(* Logix 5000 project; controller WWTP_SEC_CLX vendor 1 type 14 code 54 rev 17.2; software revision 17.00; part 2 of 13 *)
(* tags used below, declared in another part *)
   Inp_PVUncertain : BOOL;   // 1=PV Value Not Reliable, 0=OK
   Inp_Sim : BOOL;   // 1=Use simulated PV (Set_SimPV); 0=Use Input (Inp_PV)
   Cfg_NoSubstPV : BOOL;   // 1=Disallow selection of Substitute PV
   Cfg_PCmdClear : BOOL;   // 1=Clear Program Commands on receipt 0=Leave Set
   Cfg_HasHiHiAlm : BOOL;   // 1=High-High Alarm exists and will be checked
   Cfg_HasHiAlm : BOOL;   // 1=High Alarm exists and will be checked
   Cfg_HasLoAlm : BOOL;   // 1=Low Alarm exists and will be checked
   Cfg_HasLoLoAlm : BOOL;   // 1=Low-Low Alarm exists and will be checked
   Cfg_HasFailAlm : BOOL;   // 1=Analog Input Failure Alarm exists and will be checked
   Cfg_FailResetReqd : BOOL;   // 1=Reset required to clear Analog InputFailure Alarm
   Cfg_FailAckReqd : BOOL;   // 1=Acknowledge required for Analog Input Failure Alarm
   Cfg_FailSeverity : SINT;   // Failure Alarm Severity 1=info, 2=warn, 3=excep, 4=fault
   Cfg_HiHiDB : REAL;   // High-High Alarm Deadband (EU)
   Cfg_HiDB : REAL;   // High Alarm Deadband (EU)
   Cfg_LoDB : REAL;   // Low Alarm Deadband (EU)
   Cfg_LoLoDB : REAL;   // Low-Low Alarm Deadband (EU)
   Cfg_FailDB : REAL;   // Out-of-Range (fail) High/Low Deadband (EU)
   Cfg_FailMinDuration : DINT;   // Minimum time Bad or Out of Range to raise Fail Alarm (sec)
   PSet_Owner : DINT;   // Program Owner Request ID (non-zero) or Release (zero)
   PCmd_Acq : BOOL;   // Program Command to Acquire ownership (Oper to Prog)
   PCmd_Rel : BOOL;   // Program Command to Release ownership (Prog to Oper)
   PCmd_Lock : BOOL;   // Program Command to Lock Mode in Prog
   PCmd_Unlock : BOOL;   // Program Command to Unlock Mode
   PCmd_HiHiInhibit : BOOL;   // Program Command to Inhibit High-High Alarm
   PCmd_HiHiUninhibit : BOOL;   // Program Command to UninhibitHigh-High Alarm
   PCmd_HiInhibit : BOOL;   // Program Command to Inhibit High Alarm
   PCmd_HiUninhibit : BOOL;   // Program Command to Uninhibit High Alarm
   PCmd_LoInhibit : BOOL;   // Program Command to Inhibit Low Alarm
   PCmd_LoUninhibit : BOOL;   // Program Command to Uninhibit Low Alarm
   PCmd_LoLoInhibit : BOOL;   // Program Command to Inhibit Low-Low Alarm
   PCmd_LoLoUninhibit : BOOL;   // Program Command to Uninhibit Low-Low Alarm
   PCmd_FailAck : BOOL;   // Program Command to Acknowldege Analog Input Failure Alarm
   PCmd_FailInhibit : BOOL;   // Program Command to Inhibit Analog Input Failure Alarm
   PCmd_FailUninhibit : BOOL;   // Program Command to Uninhibit Analog Input Failure Alarm
   MCmd_SubstPV : BOOL;   // Maintenance Command to use Substitute PV (override input)
   MCmd_InpPV : BOOL;   // Maintenance Command to use Input PV (normal)
   Val_Owner : DINT;   // Current Object Owner ID (0=not owned)
   Sts_SubstPV : BOOL;   // 1=Using Substitute PV (Input being overridden)
   Sts_InpPV : BOOL;   // 1=Using Input PV (normal)
   Sts_PVBad : BOOL;   // 1=PV Bad quality or Out of Range
   Sts_PVUncertain : BOOL;   // 1=PV Value is Uncertain (quality)
   Err_Raw : BOOL;   // 1=Error in Config: Raw Input Scaling Min = Max
   Err_EU : BOOL;   // 1=Error in Config: Scaled EU Min = Max
   Err_Filt : BOOL;   // 1=Error in Config: PV filter params (RateTime, TC)
   Err_DB : BOOL;   // 1=Error in Config: an Alarm Deadband is < 0.0
   Err_Alarm : BOOL;   // 1=Error in Config: Invalid Alarm Min Duration or Severity
   Sts_Maint : BOOL;   // 1=Mode is Maintenance (supersedes Prog, Oper)
   Sts_Prog : BOOL;   // 1=Mode is Program
   Sts_Oper : BOOL;   // 1=Mode is Operator
   Sts_ProgOperLock : BOOL;   // 1=Program or Operator has requested Mode Lock
   Alm_HiHi : BOOL;   // 1=Analog Input is in High-High Alarm
   Ack_HiHi : BOOL;   // 1=High-High Alarm has been acknowledged
   Sts_HiHiDisabled : BOOL;   // 1=High-High Alarm is Disabled (not saved or sent)
   Sts_HiHiInhibited : BOOL;   // 1=High-High Alarm is Inhibited by logic
   Sts_HiHiSuppressed : BOOL;   // 1=High-High Alarm has been suppressed (logged only)
   Alm_Hi : BOOL;   // 1=Analog Input is in High Alarm
   Ack_Hi : BOOL;   // 1=High Alarm has been acknowledged
   Sts_HiDisabled : BOOL;   // 1=High Alarm is Disabled (not saved or sent)
   Sts_HiInhibited : BOOL;   // 1=High Alarm is Inhibited by logic
   Sts_HiSuppressed : BOOL;   // 1=High Alarm has been suppressed (logged only)
   Alm_Lo : BOOL;   // 1=Analog Input is in Low Alarm
   Ack_Lo : BOOL;   // 1=Low Alarm has been acknowledged
   Sts_LoDisabled : BOOL;   // 1=Low Alarm is Disabled (not saved or sent)
   Sts_LoInhibited : BOOL;   // 1=Low Alarm is Inhibited by logic
   Sts_LoSuppressed : BOOL;   // 1=Low Alarm has been suppressed (logged only)
   Alm_LoLo : BOOL;   // 1=Analog Input is in Low-Low Alarm
   Ack_LoLo : BOOL;   // 1=Low-Low Alarm has been acknowledged
   Sts_LoLoDisabled : BOOL;   // 1=Low-Low Alarm is Disabled (not saved or sent)
   Sts_LoLoInhibited : BOOL;   // 1=Low-Low Alarm is Inhibited by logic
   Sts_LoLoSuppressed : BOOL;   // 1=Low-Low Alarm has been suppressed (logged only)
   Sts_Fail : BOOL;   // 1=Analog Input is Out of Range or PV Bad
   Alm_Fail : BOOL;   // 1=Analog Input Failure Alarm (Bad or Out of Range)
   Ack_Fail : BOOL;   // 1=Analog Input Failure Alarm has been acknowledged
   Sts_FailDisabled : BOOL;   // 1=Analog input Failure Alarm is Disabled (not saved or sent)
   Sts_FailInhibited : BOOL;   // 1=Analog Input Failure Alarm is inhibited by logic
   Sts_FailSuppressed : BOOL;   // 1=Analog Input Failure Alarm has been suppressed (logged only)
   Rdy_SubstPV : BOOL;   // 1=Ready for MCmd_SubstPV
   Rdy_InpPV : BOOL;   // 1=Ready for MCmd_InpPV
   LoLo : P_Alarm;   // Low-Low Alarm
   Lo : P_Alarm;   // Low Alarm
   Hi : P_Alarm;   // High Alarm
   HiHi : P_Alarm;   // High-High Alarm
   Mode : P_Mode;   // Analog Input Mode Selection
   Fail : P_Alarm;   // Analog Input Failure Alarm (bad quality or out of range)
   Wrk_Notify : SINT;   // Buffer for building Val_Notify
   Wrk_SubstPV : BOOL;   // Internal flag: Using Substitute PV
   Wrk_ValidONS : BOOL;   // Selected PV goes from Infinite or Not a Number to VALID
   Wrk_SelPVInfNaN : BOOL;   // Selected PV (Input or Substitute) is Infinite or NaN
(* P_AIn, continued *)

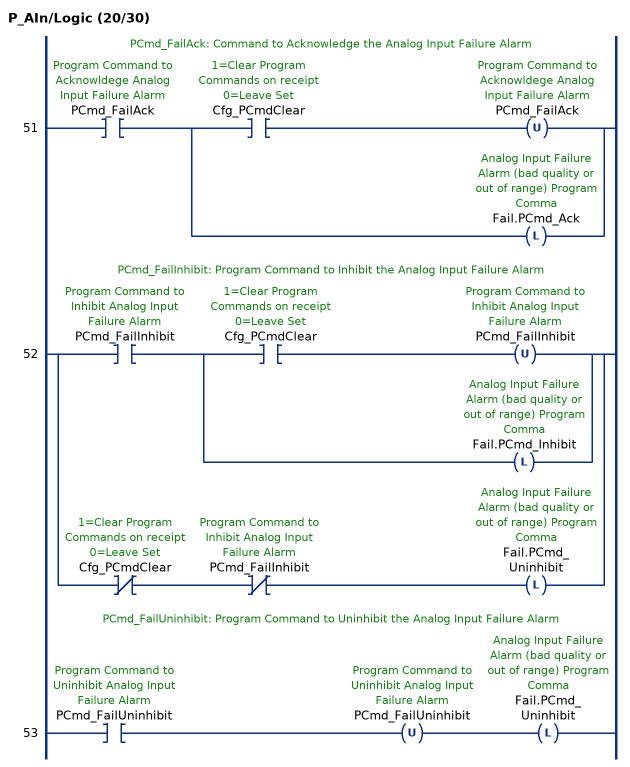
   // PCmd_FailAck: Command to Acknowledge the Analog Input Failure Alarm
   51: XIC(PCmd_FailAck)[XIC(Cfg_PCmdClear) OTU(PCmd_FailAck) ,OTL(Fail.PCmd_Ack) ];
   // PCmd_FailInhibit: Program Command to Inhibit the Analog Input Failure Alarm
   52: [XIC(PCmd_FailInhibit) [XIC(Cfg_PCmdClear) OTU(PCmd_FailInhibit) ,OTL(Fail.PCmd_Inhibit) ] ,XIO(Cfg_PCmdClear) XIO(PCmd_FailInhibit) OTL(Fail.PCmd_Uninhibit) ];
   // PCmd_FailUninhibit: Program Command to Uninhibit the Analog Input Failure Alarm
   53: XIC(PCmd_FailUninhibit)OTU(PCmd_FailUninhibit)OTL(Fail.PCmd_Uninhibit);
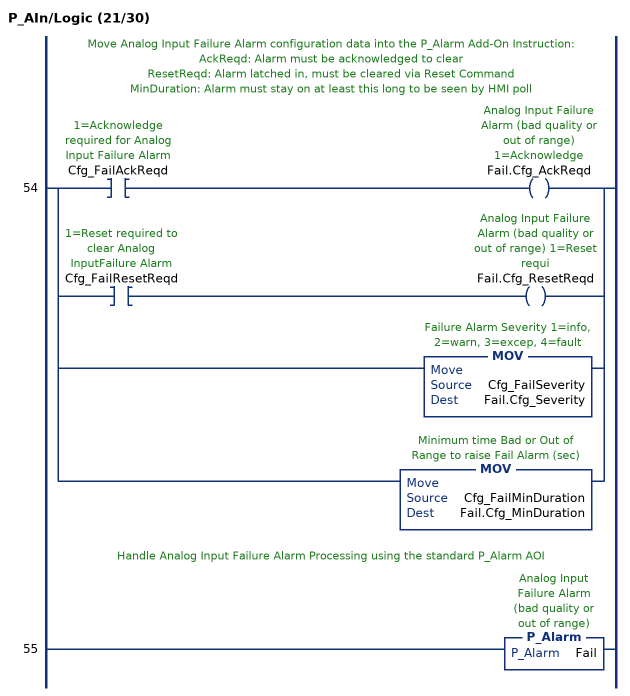
   // Move Analog Input Failure Alarm configuration data into the P_Alarm Add-On Instruction:
   // AckReqd: Alarm must be acknowledged to clear
   // ResetReqd: Alarm latched in, must be cleared via Reset Command
   // MinDuration: Alarm must stay on at least this long to be seen by HMI poll
   54: [XIC(Cfg_FailAckReqd) OTE(Fail.Cfg_AckReqd) ,XIC(Cfg_FailResetReqd) OTE(Fail.Cfg_ResetReqd) ,MOV(Cfg_FailSeverity,Fail.Cfg_Severity) ,MOV(Cfg_FailMinDuration,Fail.Cfg_MinDuration) ];
   // Handle Analog Input Failure Alarm Processing using the standard P_Alarm AOI
   55: P_Alarm(Fail);
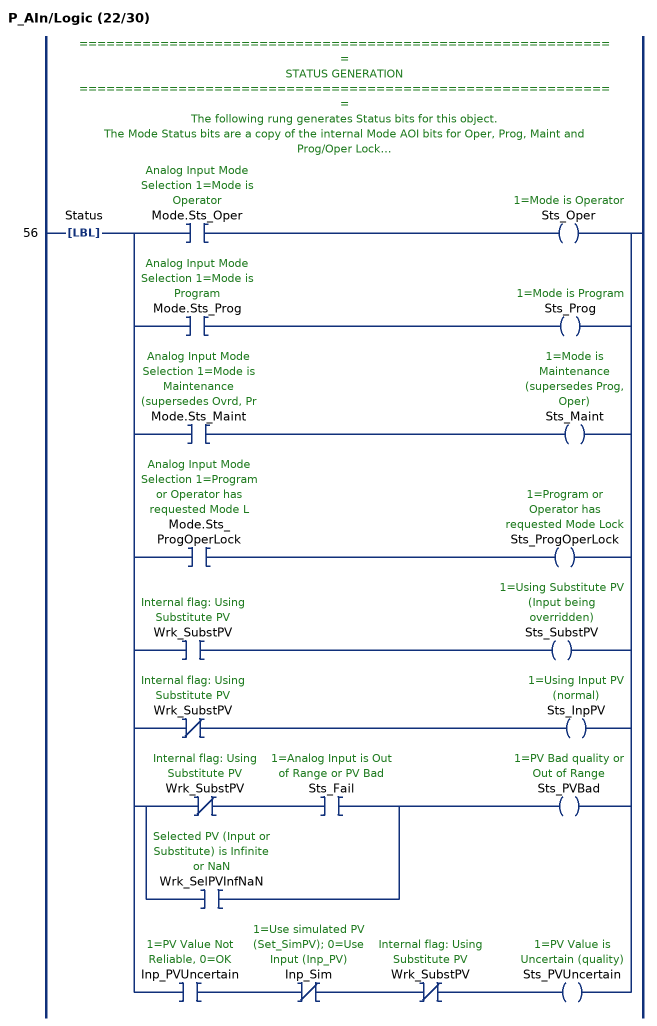
   // ============================================================
   // STATUS GENERATION
   // ============================================================
   // The following rung generates Status bits for this object.
   // The Mode Status bits are a copy of the internal Mode AOI bits for Oper, Prog, Maint and Prog/Oper Lock.
   // Remaining status bits are those not covered in the rungs above.
   56: LBL(Status)[XIC(Mode.Sts_Oper) OTE(Sts_Oper) ,XIC(Mode.Sts_Prog) OTE(Sts_Prog) ,XIC(Mode.Sts_Maint) OTE(Sts_Maint) ,XIC(Mode.Sts_ProgOperLock) OTE(Sts_ProgOperLock) ,XIC(Wrk_SubstPV) OTE(Sts_SubstPV) ,XIO(Wrk_SubstPV) OTE(Sts_InpPV) ,[XIO(Wrk_SubstPV) XIC(Sts_Fail) ,XIC(Wrk_SelPVInfNaN) ] OTE(Sts_PVBad) ,XIC(Inp_PVUncertain) XIO(Inp_Sim) XIO(Wrk_SubstPV) OTE(Sts_PVUncertain) ];
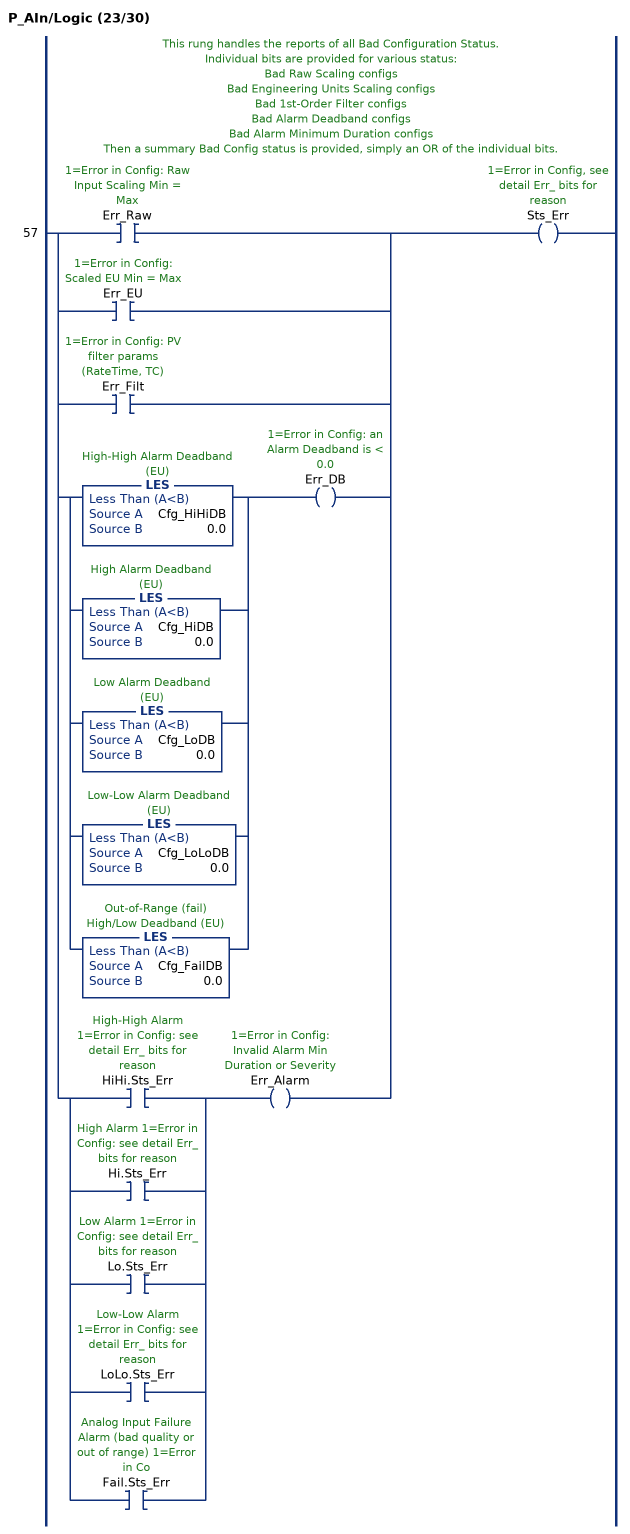
   // This rung handles the reports of all Bad Configuration Status.
   // Individual bits are provided for various status:
   // Bad Raw Scaling configs
   // Bad Engineering Units Scaling configs
   // Bad 1st-Order Filter configs
   // Bad Alarm Deadband configs
   // Bad Alarm Minimum Duration configs
   // Then a summary Bad Config status is provided, simply an OR of the individual bits.
   57: [XIC(Err_Raw) ,XIC(Err_EU) ,XIC(Err_Filt) ,[LES(Cfg_HiHiDB,0.0) ,LES(Cfg_HiDB,0.0) ,LES(Cfg_LoDB,0.0) ,LES(Cfg_LoLoDB,0.0) ,LES(Cfg_FailDB,0.0) ] OTE(Err_DB) ,[XIC(HiHi.Sts_Err) ,XIC(Hi.Sts_Err) ,XIC(Lo.Sts_Err) ,XIC(LoLo.Sts_Err) ,XIC(Fail.Sts_Err) ] OTE(Err_Alarm) ]OTE(Sts_Err);
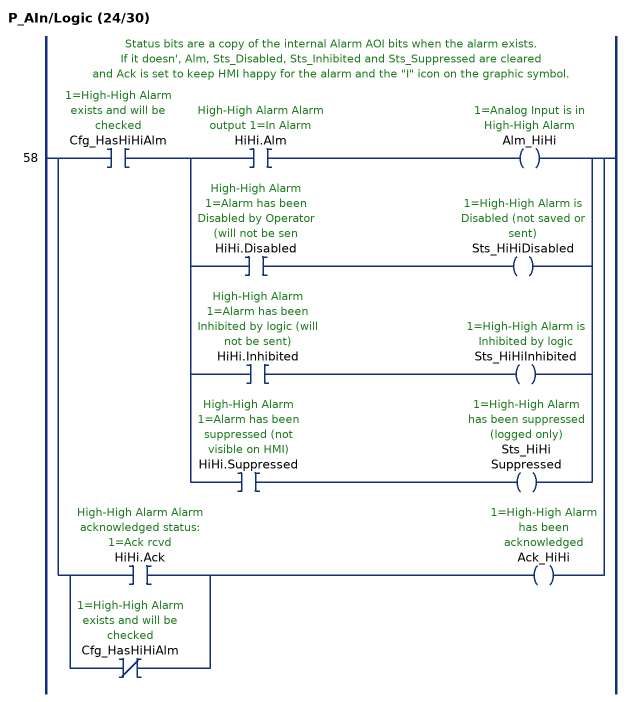
   // Status bits are a copy of the internal Alarm AOI bits when the alarm exists.
   // If it doesn', Alm, Sts_Disabled, Sts_Inhibited and Sts_Suppressed are cleared
   // and Ack is set to keep HMI happy for the alarm and the "I" icon on the graphic symbol.
   58: [XIC(Cfg_HasHiHiAlm) [XIC(HiHi.Alm) OTE(Alm_HiHi) ,XIC(HiHi.Disabled) OTE(Sts_HiHiDisabled) ,XIC(HiHi.Inhibited) OTE(Sts_HiHiInhibited) ,XIC(HiHi.Suppressed) OTE(Sts_HiHiSuppressed) ] ,[XIC(HiHi.Ack) ,XIO(Cfg_HasHiHiAlm) ] OTE(Ack_HiHi) ];
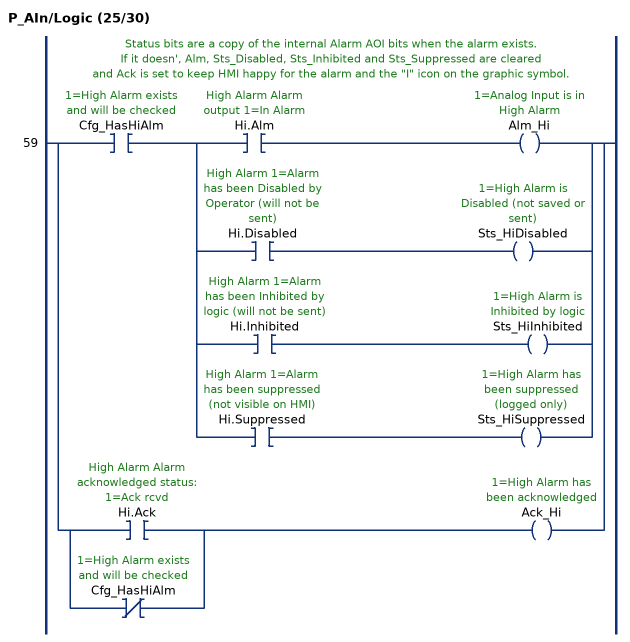
   // Status bits are a copy of the internal Alarm AOI bits when the alarm exists.
   // If it doesn', Alm, Sts_Disabled, Sts_Inhibited and Sts_Suppressed are cleared
   // and Ack is set to keep HMI happy for the alarm and the "I" icon on the graphic symbol.
   59: [XIC(Cfg_HasHiAlm) [XIC(Hi.Alm) OTE(Alm_Hi) ,XIC(Hi.Disabled) OTE(Sts_HiDisabled) ,XIC(Hi.Inhibited) OTE(Sts_HiInhibited) ,XIC(Hi.Suppressed) OTE(Sts_HiSuppressed) ] ,[XIC(Hi.Ack) ,XIO(Cfg_HasHiAlm) ] OTE(Ack_Hi) ];
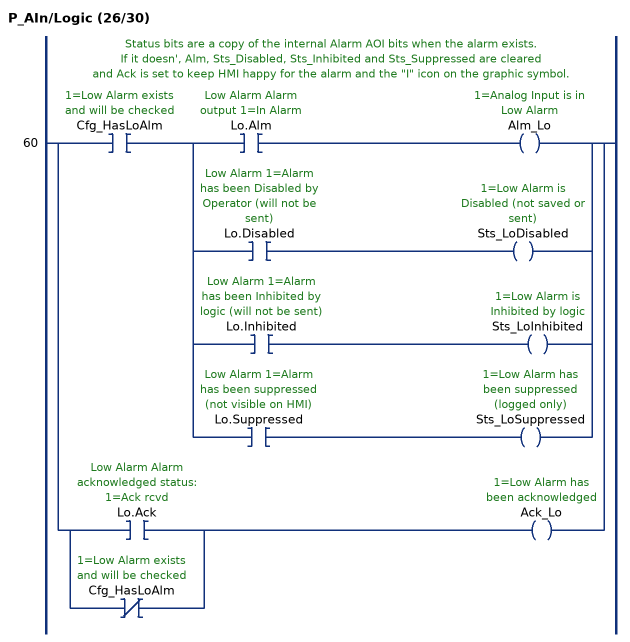
   // Status bits are a copy of the internal Alarm AOI bits when the alarm exists.
   // If it doesn', Alm, Sts_Disabled, Sts_Inhibited and Sts_Suppressed are cleared
   // and Ack is set to keep HMI happy for the alarm and the "I" icon on the graphic symbol.
   60: [XIC(Cfg_HasLoAlm) [XIC(Lo.Alm) OTE(Alm_Lo) ,XIC(Lo.Disabled) OTE(Sts_LoDisabled) ,XIC(Lo.Inhibited) OTE(Sts_LoInhibited) ,XIC(Lo.Suppressed) OTE(Sts_LoSuppressed) ] ,[XIC(Lo.Ack) ,XIO(Cfg_HasLoAlm) ] OTE(Ack_Lo) ];
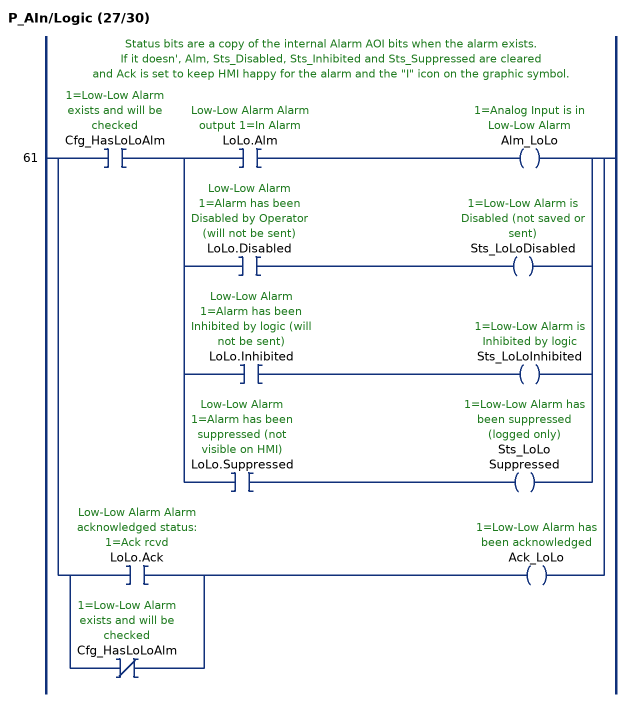
   // Status bits are a copy of the internal Alarm AOI bits when the alarm exists.
   // If it doesn', Alm, Sts_Disabled, Sts_Inhibited and Sts_Suppressed are cleared
   // and Ack is set to keep HMI happy for the alarm and the "I" icon on the graphic symbol.
   61: [XIC(Cfg_HasLoLoAlm) [XIC(LoLo.Alm) OTE(Alm_LoLo) ,XIC(LoLo.Disabled) OTE(Sts_LoLoDisabled) ,XIC(LoLo.Inhibited) OTE(Sts_LoLoInhibited) ,XIC(LoLo.Suppressed) OTE(Sts_LoLoSuppressed) ] ,[XIC(LoLo.Ack) ,XIO(Cfg_HasLoLoAlm) ] OTE(Ack_LoLo) ];
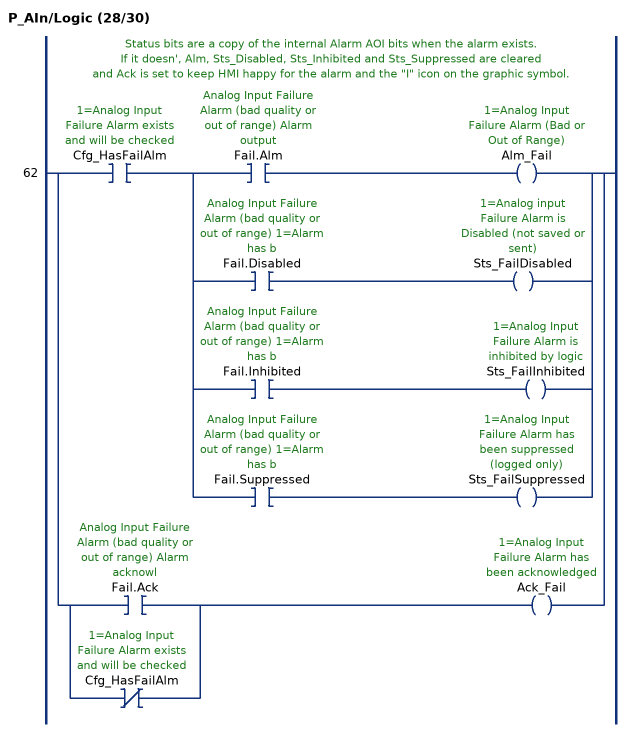
   // Status bits are a copy of the internal Alarm AOI bits when the alarm exists.
   // If it doesn', Alm, Sts_Disabled, Sts_Inhibited and Sts_Suppressed are cleared
   // and Ack is set to keep HMI happy for the alarm and the "I" icon on the graphic symbol.
   62: [XIC(Cfg_HasFailAlm) [XIC(Fail.Alm) OTE(Alm_Fail) ,XIC(Fail.Disabled) OTE(Sts_FailDisabled) ,XIC(Fail.Inhibited) OTE(Sts_FailInhibited) ,XIC(Fail.Suppressed) OTE(Sts_FailSuppressed) ] ,[XIC(Fail.Ack) ,XIO(Cfg_HasFailAlm) ] OTE(Ack_Fail) ];
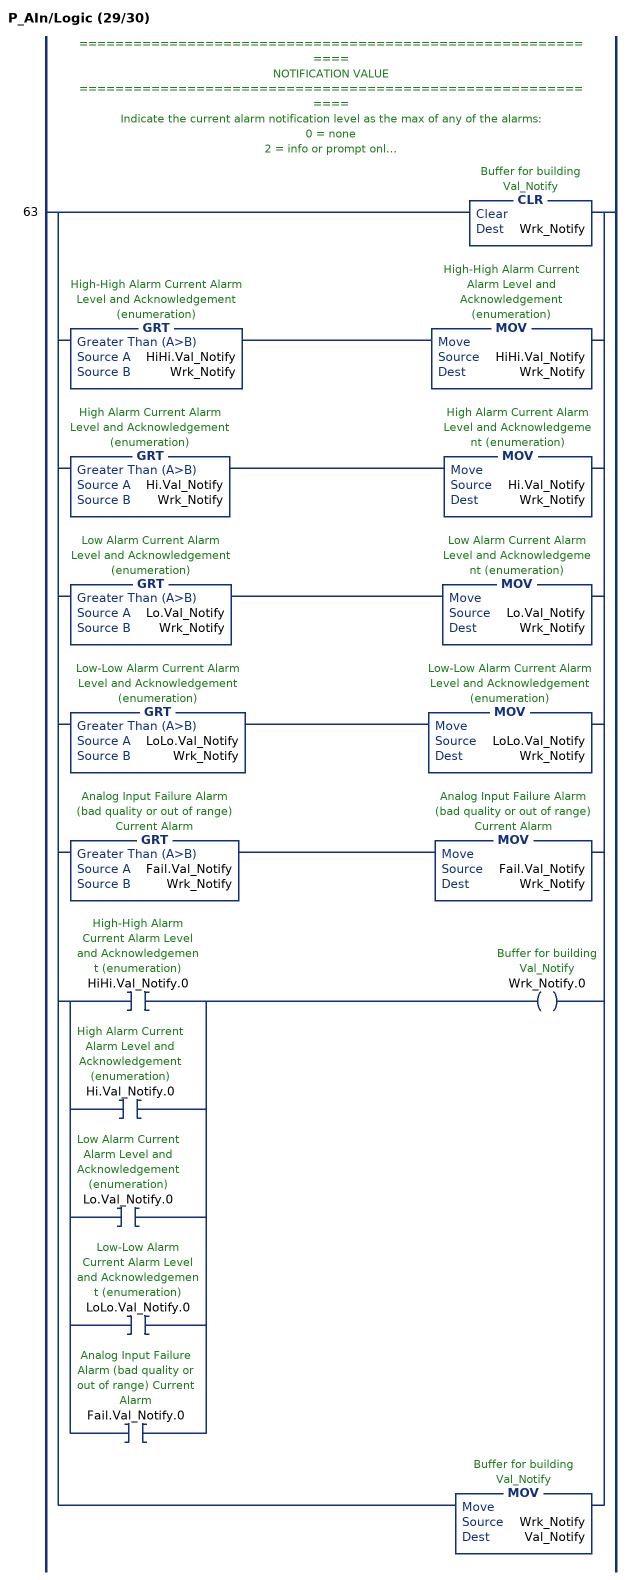
   // ============================================================
   // NOTIFICATION VALUE
   // ============================================================
   // Indicate the current alarm notification level as the max of any of the alarms:
   // 0 = none
   // 2 = info or prompt only
   // 4 = warning
   // 6 = exception (equipment impact)
   // 8 = fault (equipment failure)
   // Add one for any unsuppressed alarm that is not acknowledged (for blink).
   63: [CLR(Wrk_Notify) ,GRT(HiHi.Val_Notify,Wrk_Notify) MOV(HiHi.Val_Notify,Wrk_Notify) ,GRT(Hi.Val_Notify,Wrk_Notify) MOV(Hi.Val_Notify,Wrk_Notify) ,GRT(Lo.Val_Notify,Wrk_Notify) MOV(Lo.Val_Notify,Wrk_Notify) ,GRT(LoLo.Val_Notify,Wrk_Notify) MOV(LoLo.Val_Notify,Wrk_Notify) ,GRT(Fail.Val_Notify,Wrk_Notify) MOV(Fail.Val_Notify,Wrk_Notify) ,[XIC(HiHi.Val_Notify.0) ,XIC(Hi.Val_Notify.0) ,XIC(Lo.Val_Notify.0) ,XIC(LoLo.Val_Notify.0) ,XIC(Fail.Val_Notify.0) ] OTE(Wrk_Notify.0) ,MOV(Wrk_Notify,Val_Notify) ];
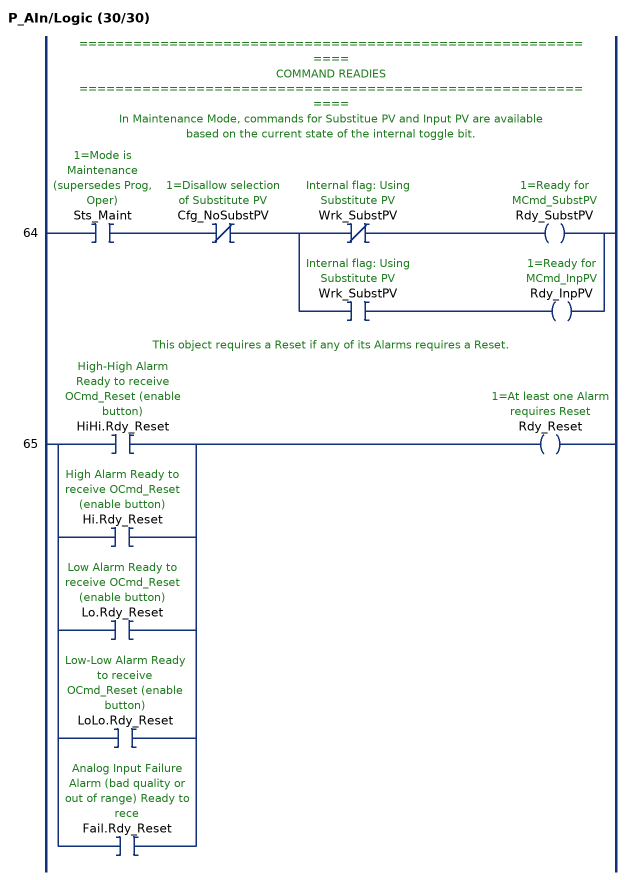
   // ============================================================
   // COMMAND READIES
   // ============================================================
   // In Maintenance Mode, commands for Substitue PV and Input PV are available
   // based on the current state of the internal toggle bit.
   64: XIC(Sts_Maint)XIO(Cfg_NoSubstPV)[XIO(Wrk_SubstPV) OTE(Rdy_SubstPV) ,XIC(Wrk_SubstPV) OTE(Rdy_InpPV) ];
   // This object requires a Reset if any of its Alarms requires a Reset.
   65: [XIC(HiHi.Rdy_Reset) ,XIC(Hi.Rdy_Reset) ,XIC(Lo.Rdy_Reset) ,XIC(LoLo.Rdy_Reset) ,XIC(Fail.Rdy_Reset) ]OTE(Rdy_Reset);
END_ROUTINE

ROUTINE Prescan   (* ladder *)
// Clear Ownership. clear "lurking" Commands
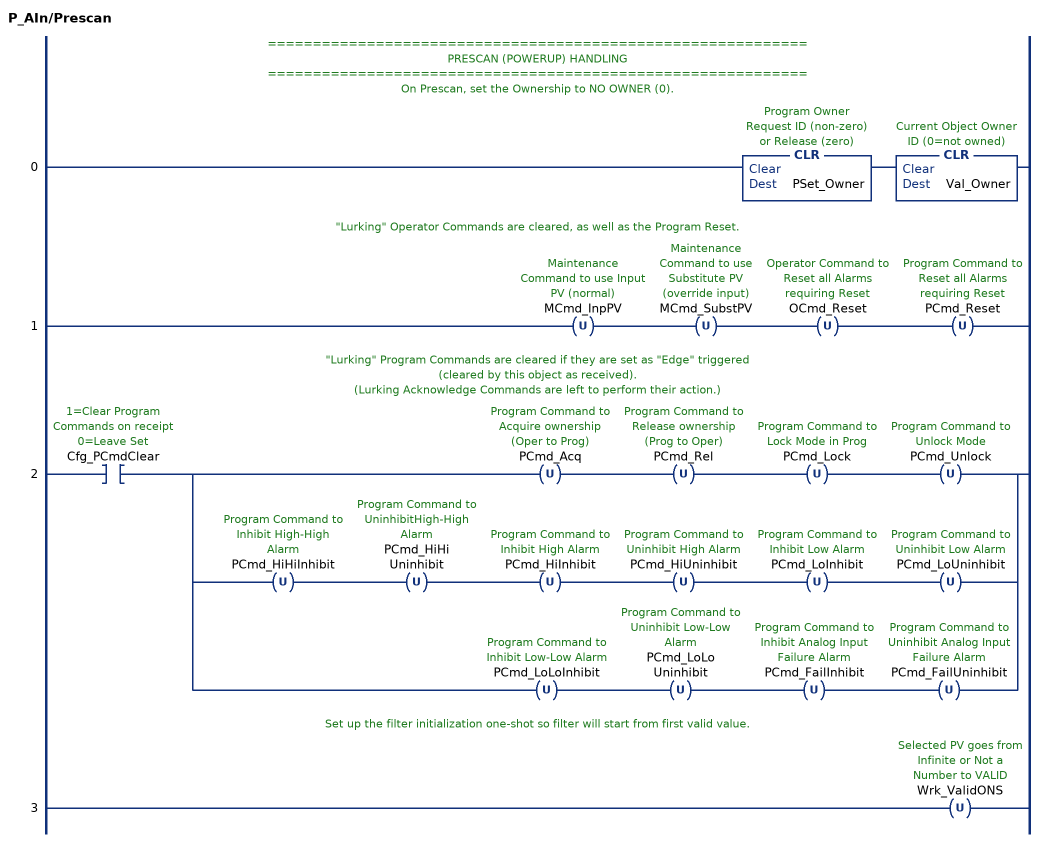
   // ============================================================
   // PRESCAN (POWERUP) HANDLING
   // ============================================================
   // On Prescan, set the Ownership to NO OWNER (0).
   0: CLR(PSet_Owner)CLR(Val_Owner);
   // "Lurking" Operator Commands are cleared, as well as the Program Reset.
   1: OTU(MCmd_InpPV)OTU(MCmd_SubstPV)OTU(OCmd_Reset)OTU(PCmd_Reset);
   // "Lurking" Program Commands are cleared if they are set as "Edge" triggered
   // (cleared by this object as received).
   // (Lurking Acknowledge Commands are left to perform their action.)
   2: XIC(Cfg_PCmdClear)[OTU(PCmd_Acq) OTU(PCmd_Rel) OTU(PCmd_Lock) OTU(PCmd_Unlock) ,OTU(PCmd_HiHiInhibit) OTU(PCmd_HiHiUninhibit) OTU(PCmd_HiInhibit) OTU(PCmd_HiUninhibit) OTU(PCmd_LoInhibit) OTU(PCmd_LoUninhibit) ,OTU(PCmd_LoLoInhibit) OTU(PCmd_LoLoUninhibit) OTU(PCmd_FailInhibit) OTU(PCmd_FailUninhibit) ];
   // Set up the filter initialization one-shot so filter will start from first valid value.
   3: OTU(Wrk_ValidONS);
END_ROUTINE
END_ADD_ON_INSTRUCTION

ADD_ON_INSTRUCTION P_Alarm   (* revision 0.21, ExecutePrescan, ExecuteEnableInFalse *)
// Alarm
// Revision note:
// Fixed differences between Logic and EnableInFalse; fixed scan order dependency.
// Help:
// This instruction monitors one input condition and provides one Alarm with:
//   * configurable Alarm delay, latching, acknowledgement, and severity
//   * commands for enable/disable (oper) and inhibit/uninhibit (prog)
//   * FTA&E suppress/unsuppress support
// This instruction is usually nested within other instructions, with one instance used for each Alarm generated by the containing instruction.  It may also be used as a standalone instruction for Alarm conditions generated by custom logic.
VAR_INPUT
   Inp : BOOL := 1; {visible}   // Alarm Condition Input 1=Alarm
   Inp_Reset : BOOL; {visible}   // 1=Reset Alarm requiring reset
   Cfg_ResetReqd : BOOL;   // 1=Reset required to clear Alarm
   Cfg_AckReqd : BOOL := 1;   // 1=Acknowledge required for Alarm
   Cfg_Severity : SINT := 3;   // 1=Info Only; 2=Warning; 3=Process Exception; 4=Fault
   Cfg_MinDuration : DINT;   // Minimum time (sec) Input must stay on to generate Alarm
   PCmd_Reset : BOOL;   // Program Command to Reset latched alarm
   PCmd_Ack : BOOL;   // Program Command to Acknowledge alarm
   PCmd_Inhibit : BOOL;   // Program Command to Inhibit alarm (force Alm to 0)
   PCmd_Uninhibit : BOOL;   // Program Command to Uninhibit alarm
   OCmd_Reset : BOOL;   // Operator Command to Reset latched alarm
   OCmd_Ack : BOOL;   // Operator Command to Acknowledge alarm
   OCmd_Disable : BOOL;   // Operator Command to Disable alarm (force Alm to 0)
   OCmd_Enable : BOOL;   // Operator Command to Enable alarm
END_VAR
VAR_OUTPUT
   Val_Notify : SINT;   // Current Alarm Level and Acknowledgement (enumeration)
   Alm : BOOL; {visible}   // Alarm output 1=In Alarm
   Ack : BOOL := 1; {visible}   // Alarm acknowledged status: 1=Ack rcvd
   Disabled : BOOL; {visible}   // 1=Alarm has been Disabled by Operator (will not be sent)
   Inhibited : BOOL; {visible}   // 1=Alarm has been Inhibited by logic (will not be sent)
   Suppressed : BOOL; {visible}   // 1=Alarm has been suppressed (not visible on HMI)
   Sts_Err : BOOL;   // 1=Error in Config: see detail Err_ bits for reason
   Err_MinDuration : BOOL;   // 1=Error in Config: Invalid Min Duration (use 0 to 2147483)
   Err_Severity : BOOL;   // 1=Error in Config: Invalid Severity (use 1 to 4)
   Rdy_Reset : BOOL;   // Ready to receive OCmd_Reset (enable button)
   Rdy_Ack : BOOL;   // Ready to receive OCmd_Ack (enable button)
   Rdy_Disable : BOOL := 1;   // Ready to receive OCmd_Disable (enable button)
   Rdy_Enable : BOOL;   // Ready to receive OCmd_Enable (enable button)
END_VAR
VAR
   Wrk_MinDurationT : TIMER;   // Alarm Condition Minimum Duration Timer
   Wrk_Alm : BOOL;   // Internal Alarm Status
   Wrk_Inhibited : BOOL;   // Internal Alarm Inhibit Status
   Wrk_AlmMinOnT : TIMER := (PRE := 5000);   // Alarm output minimum ON time to be seen by alarm server
END_VAR

ROUTINE EnableInFalse   (* ladder *)
// Perform Alarm processing, but Invert Alarm Input ("Inp") for use on LD rung (EnableIn False)
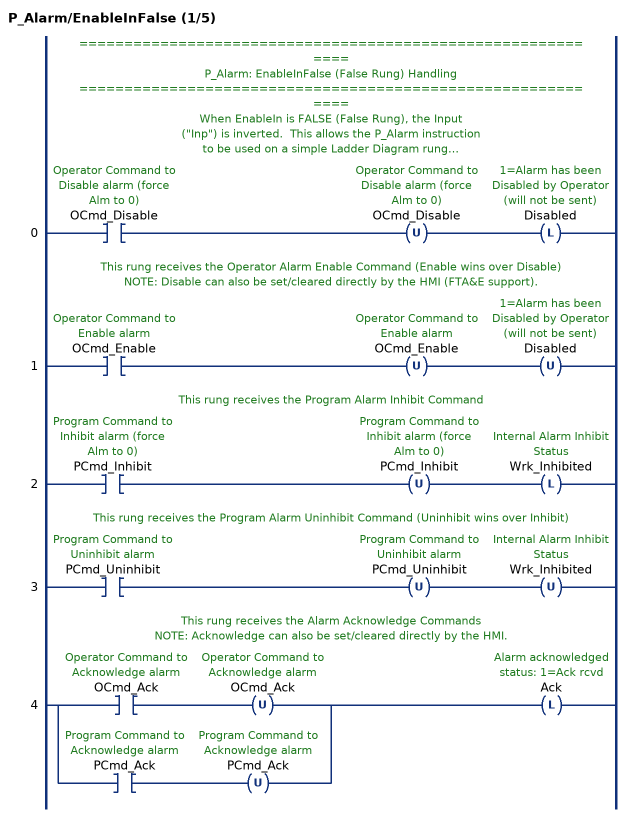
   // ============================================================
   // P_Alarm: EnableInFalse (False Rung) Handling
   // ============================================================
   // When EnableIn is FALSE (False Rung), the Input
   // ("Inp") is inverted.  This allows the P_Alarm instruction
   // to be used on a simple Ladder Diagram rung:
   // XIC  (condition)   P_Alarm (Alarm)
   // All processing is identical to the normal Logic
   // routine, except references to Inp are inverted!
   // ============================================================
   // COMMAND PROCESSING
   // ============================================================
   // These rungs handle received Commands:
   // Operator Commands (OCmd_xx) from the HMI and
   // Program Command (PCmd_xx) from other objects.
   // NOTE:  ALARM COMMANDS ARE ACCEPTED REGARDLESS OF MODE.
   // This rung receives the Operator Alarm Disable Command
   0: XIC(OCmd_Disable)OTU(OCmd_Disable)OTL(Disabled);
   // This rung receives the Operator Alarm Enable Command (Enable wins over Disable)
   // NOTE: Disable can also be set/cleared directly by the HMI (FTA&E support).
   1: XIC(OCmd_Enable)OTU(OCmd_Enable)OTU(Disabled);
   // This rung receives the Program Alarm Inhibit Command
   2: XIC(PCmd_Inhibit)OTU(PCmd_Inhibit)OTL(Wrk_Inhibited);
   // This rung receives the Program Alarm Uninhibit Command (Uninhibit wins over Inhibit)
   3: XIC(PCmd_Uninhibit)OTU(PCmd_Uninhibit)OTU(Wrk_Inhibited);
   // This rung receives the Alarm Acknowledge Commands
   // NOTE: Acknowledge can also be set/cleared directly by the HMI.
   4: [XIC(OCmd_Ack) OTU(OCmd_Ack) ,XIC(PCmd_Ack) OTU(PCmd_Ack) ]OTL(Ack);
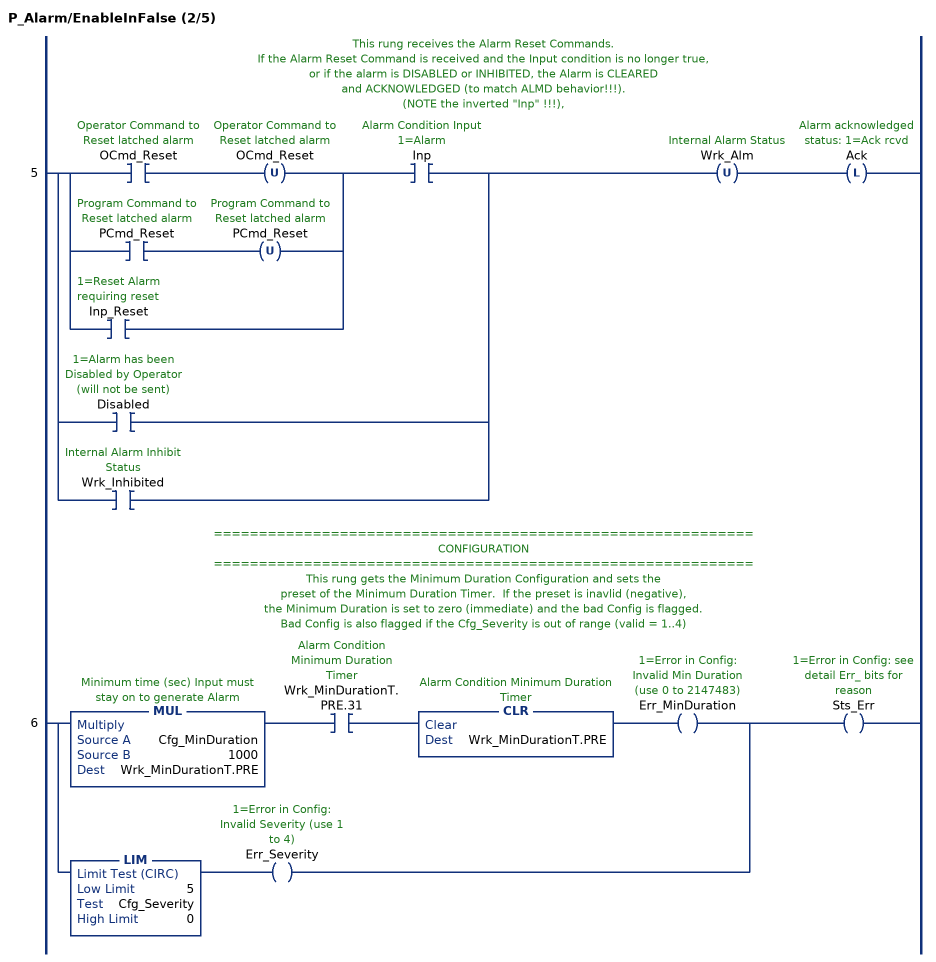
   // This rung receives the Alarm Reset Commands.
   // If the Alarm Reset Command is received and the Input condition is no longer true,
   // or if the alarm is DISABLED or INHIBITED, the Alarm is CLEARED
   // and ACKNOWLEDGED (to match ALMD behavior!!!).
   // (NOTE the inverted "Inp" !!!),
   5: [[XIC(OCmd_Reset) OTU(OCmd_Reset) ,XIC(PCmd_Reset) OTU(PCmd_Reset) ,XIC(Inp_Reset) ] XIC(Inp) ,XIC(Disabled) ,XIC(Wrk_Inhibited) ]OTU(Wrk_Alm)OTL(Ack);
   // ============================================================
   // CONFIGURATION
   // ============================================================
   // This rung gets the Minimum Duration Configuration and sets the
   // preset of the Minimum Duration Timer.  If the preset is inavlid (negative),
   // the Minimum Duration is set to zero (immediate) and the bad Config is flagged.
   // Bad Config is also flagged if the Cfg_Severity is out of range (valid = 1..4)
   6: [MUL(Cfg_MinDuration,1000,Wrk_MinDurationT.PRE) XIC(Wrk_MinDurationT.PRE.31) CLR(Wrk_MinDurationT.PRE) OTE(Err_MinDuration) ,LIM(5,Cfg_Severity,0) OTE(Err_Severity) ]OTE(Sts_Err);
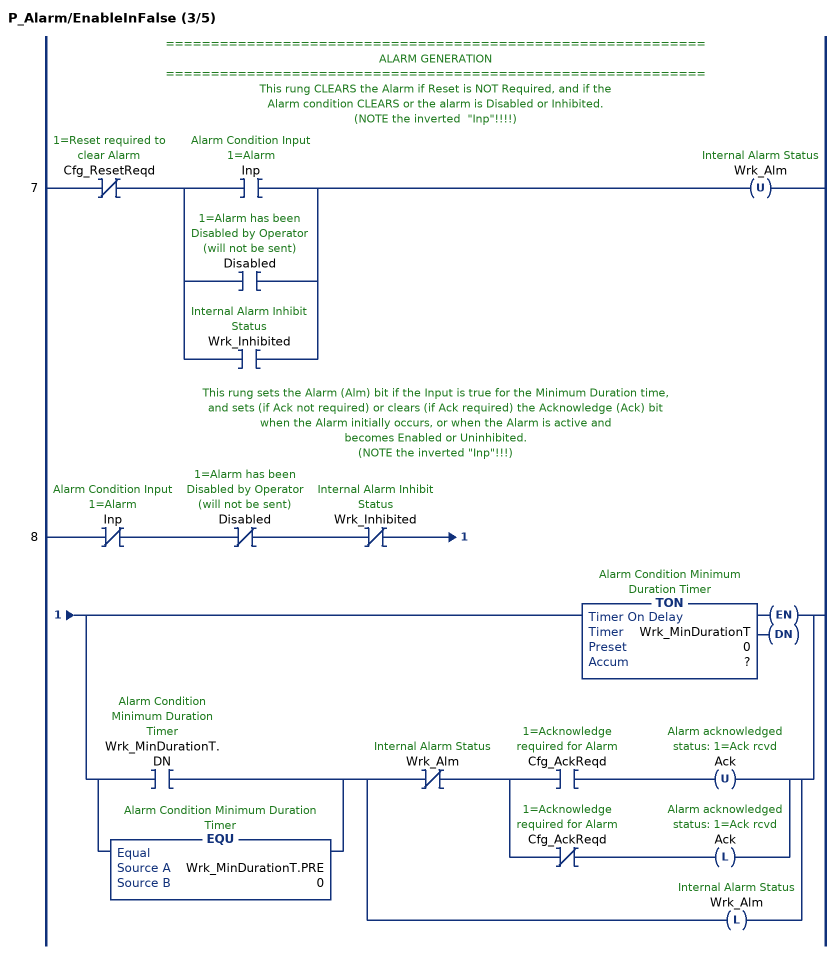
   // ============================================================
   // ALARM GENERATION
   // ============================================================
   // This rung CLEARS the Alarm if Reset is NOT Required, and if the
   // Alarm condition CLEARS or the alarm is Disabled or Inhibited.
   // (NOTE the inverted  "Inp"!!!!)
   7: XIO(Cfg_ResetReqd)[XIC(Inp) ,XIC(Disabled) ,XIC(Wrk_Inhibited) ]OTU(Wrk_Alm);
   // This rung sets the Alarm (Alm) bit if the Input is true for the Minimum Duration time,
   // and sets (if Ack not required) or clears (if Ack required) the Acknowledge (Ack) bit
   // when the Alarm initially occurs, or when the Alarm is active and
   // becomes Enabled or Uninhibited.
   // (NOTE the inverted "Inp"!!!)
   8: XIO(Inp)XIO(Disabled)XIO(Wrk_Inhibited)[TON(Wrk_MinDurationT,?,?) ,[XIC(Wrk_MinDurationT.DN) ,EQU(Wrk_MinDurationT.PRE,0) ] [XIO(Wrk_Alm) [XIC(Cfg_AckReqd) OTU(Ack) ,XIO(Cfg_AckReqd) OTL(Ack) ] ,OTL(Wrk_Alm) ] ];
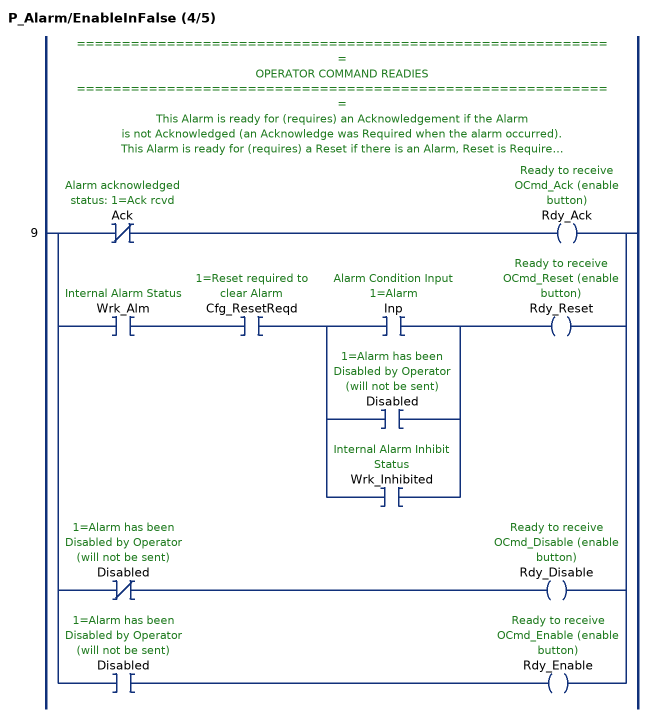
   // ============================================================
   // OPERATOR COMMAND READIES
   // ============================================================
   // This Alarm is ready for (requires) an Acknowledgement if the Alarm
   // is not Acknowledged (an Acknowledge was Required when the alarm occurred).
   // This Alarm is ready for (requires) a Reset if there is an Alarm, Reset is Required
   // and the Alarm Condition is CLEARED
   // (NOTE the inverted "Inp"!!!)
   // If the Alarm is NOT Disabled, it is ready for Disable.
   // If the Alarm IS Disabled, it is ready for Enable.
   9: [XIO(Ack) OTE(Rdy_Ack) ,XIC(Wrk_Alm) XIC(Cfg_ResetReqd) [XIC(Inp) ,XIC(Disabled) ,XIC(Wrk_Inhibited) ] OTE(Rdy_Reset) ,XIO(Disabled) OTE(Rdy_Disable) ,XIC(Disabled) OTE(Rdy_Enable) ];
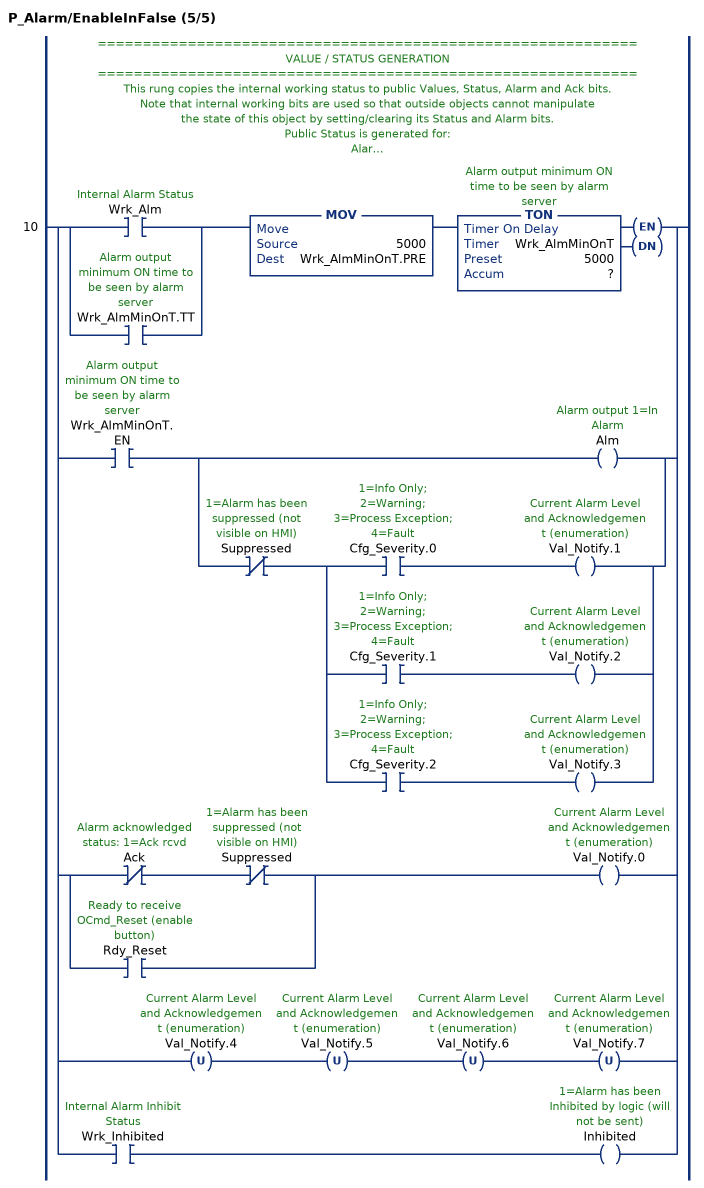
   // ============================================================
   // VALUE / STATUS GENERATION
   // ============================================================
   // This rung copies the internal working status to public Values, Status, Alarm and Ack bits.
   // Note that internal working bits are used so that outside objects cannot manipulate
   // the state of this object by setting/clearing its Status and Alarm bits.
   // Public Status is generated for:
   // Alarm
   // Notify Level (color, blink)
   // Alarm Inhibited
   // (Ack, Suppressed and Disabled can be set/cleared by the HMI directly.)
   10: [[XIC(Wrk_Alm) ,XIC(Wrk_AlmMinOnT.TT) ] MOV(5000,Wrk_AlmMinOnT.PRE) TON(Wrk_AlmMinOnT,?,?) ,XIC(Wrk_AlmMinOnT.EN) [OTE(Alm) ,XIO(Suppressed) [XIC(Cfg_Severity.0) OTE(Val_Notify.1) ,XIC(Cfg_Severity.1) OTE(Val_Notify.2) ,XIC(Cfg_Severity.2) OTE(Val_Notify.3) ] ] ,[XIO(Ack) XIO(Suppressed) ,XIC(Rdy_Reset) ] OTE(Val_Notify.0) ,OTU(Val_Notify.4) OTU(Val_Notify.5) OTU(Val_Notify.6) OTU(Val_Notify.7) ,XIC(Wrk_Inhibited) OTE(Inhibited) ];
END_ROUTINE

ROUTINE Logic   (* ladder *)
// Perform Alarm processing: delay, latch/reset, acknowledge, enable/disable, inhibit/uninhibit, suppress/unsuppress
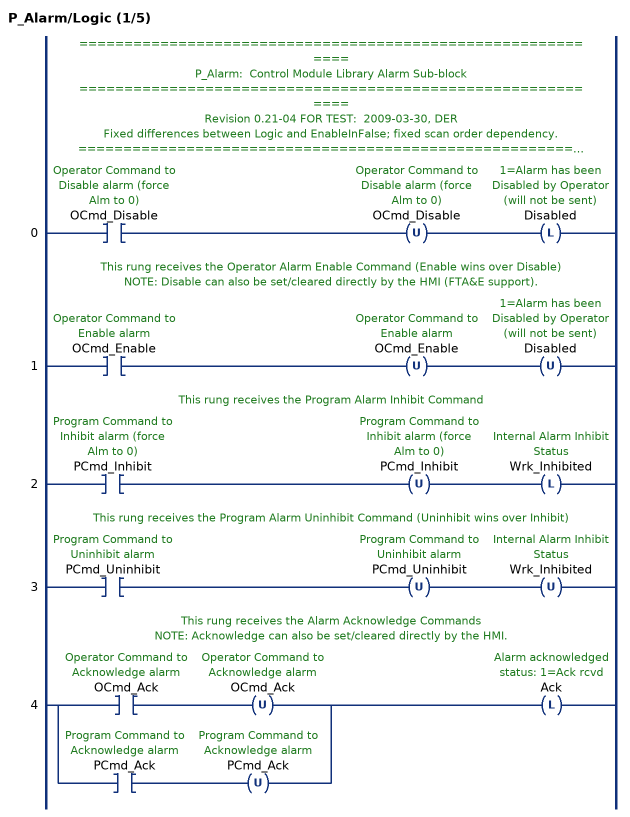
   // ============================================================
   // P_Alarm:  Control Module Library Alarm Sub-block
   // ============================================================
   // Revision 0.21-04 FOR TEST:  2009-03-30, DER
   // Fixed differences between Logic and EnableInFalse; fixed scan order dependency.
   // ============================================================
   // This instruction provides standard Alarm handling for a given input Alarm condition.
   // This instruction should be imbedded in any instruction that generates alarms,
   // one instance per alarm generated.
   // ============================================================
   // POWERUP / INVALID STATE HANDLING
   // ============================================================
   // All internal Work (state) bits maintain states through a power cycle and are
   // independent.  No first-scan logic is required.  See the Prescan routine for
   // powerup / prescan code.
   // ============================================================
   // COMMAND PROCESSING
   // ============================================================
   // These rungs handle received Commands:
   // Operator Commands (OCmd_xx) from the HMI and
   // Program Command (PCmd_xx) from other objects.
   // NOTE:  ALARM COMMANDS ARE ACCEPTED REGARDLESS OF MODE.
   // This rung receives the Operator Alarm Disable Command
   0: XIC(OCmd_Disable)OTU(OCmd_Disable)OTL(Disabled);
   // This rung receives the Operator Alarm Enable Command (Enable wins over Disable)
   // NOTE: Disable can also be set/cleared directly by the HMI (FTA&E support).
   1: XIC(OCmd_Enable)OTU(OCmd_Enable)OTU(Disabled);
   // This rung receives the Program Alarm Inhibit Command
   2: XIC(PCmd_Inhibit)OTU(PCmd_Inhibit)OTL(Wrk_Inhibited);
   // This rung receives the Program Alarm Uninhibit Command (Uninhibit wins over Inhibit)
   3: XIC(PCmd_Uninhibit)OTU(PCmd_Uninhibit)OTU(Wrk_Inhibited);
   // This rung receives the Alarm Acknowledge Commands
   // NOTE: Acknowledge can also be set/cleared directly by the HMI.
   4: [XIC(OCmd_Ack) OTU(OCmd_Ack) ,XIC(PCmd_Ack) OTU(PCmd_Ack) ]OTL(Ack);
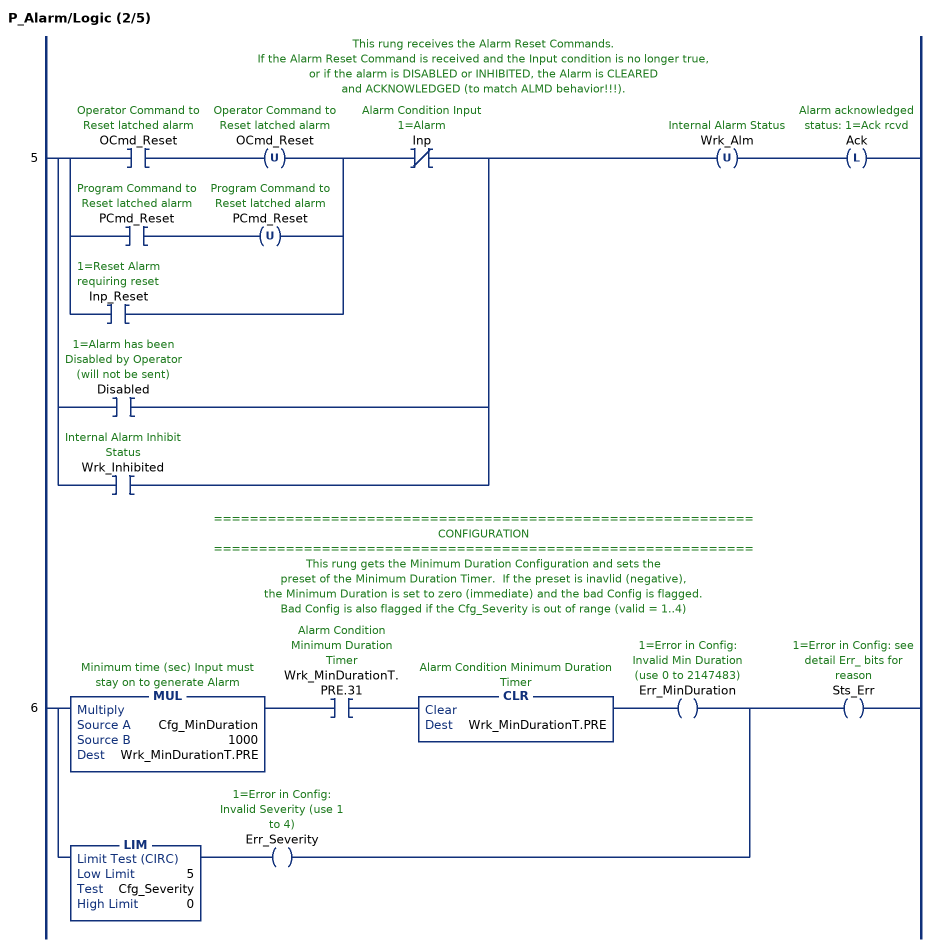
   // This rung receives the Alarm Reset Commands.
   // If the Alarm Reset Command is received and the Input condition is no longer true,
   // or if the alarm is DISABLED or INHIBITED, the Alarm is CLEARED
   // and ACKNOWLEDGED (to match ALMD behavior!!!).
   5: [[XIC(OCmd_Reset) OTU(OCmd_Reset) ,XIC(PCmd_Reset) OTU(PCmd_Reset) ,XIC(Inp_Reset) ] XIO(Inp) ,XIC(Disabled) ,XIC(Wrk_Inhibited) ]OTU(Wrk_Alm)OTL(Ack);
   // ============================================================
   // CONFIGURATION
   // ============================================================
   // This rung gets the Minimum Duration Configuration and sets the
   // preset of the Minimum Duration Timer.  If the preset is inavlid (negative),
   // the Minimum Duration is set to zero (immediate) and the bad Config is flagged.
   // Bad Config is also flagged if the Cfg_Severity is out of range (valid = 1..4)
   6: [MUL(Cfg_MinDuration,1000,Wrk_MinDurationT.PRE) XIC(Wrk_MinDurationT.PRE.31) CLR(Wrk_MinDurationT.PRE) OTE(Err_MinDuration) ,LIM(5,Cfg_Severity,0) OTE(Err_Severity) ]OTE(Sts_Err);
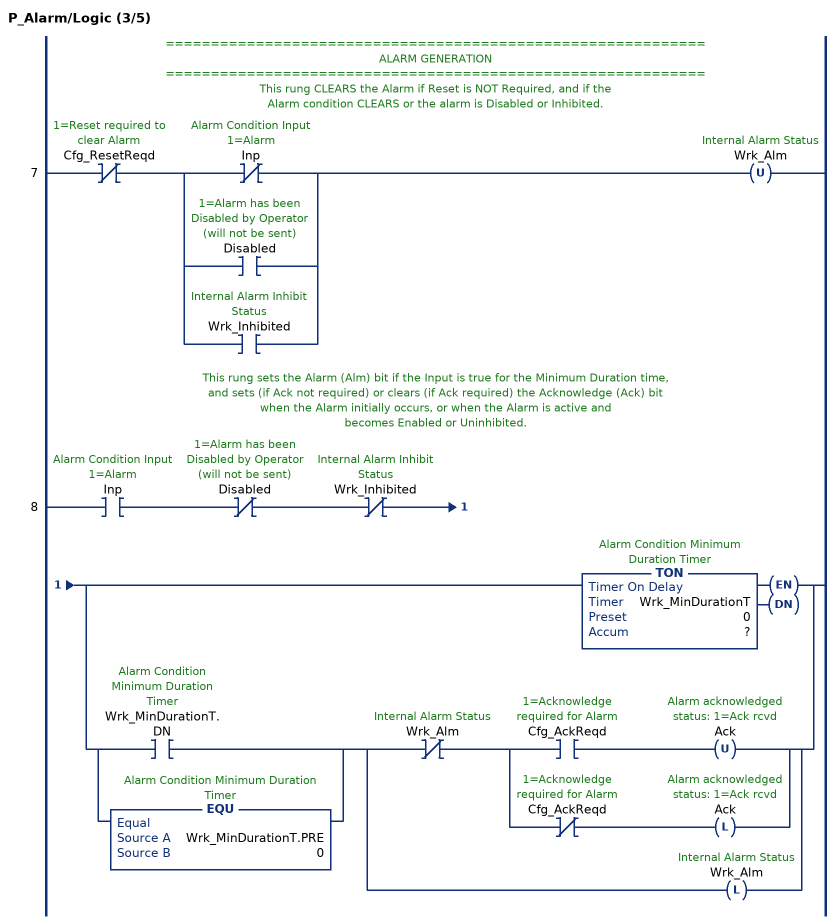
   // ============================================================
   // ALARM GENERATION
   // ============================================================
   // This rung CLEARS the Alarm if Reset is NOT Required, and if the
   // Alarm condition CLEARS or the alarm is Disabled or Inhibited.
   7: XIO(Cfg_ResetReqd)[XIO(Inp) ,XIC(Disabled) ,XIC(Wrk_Inhibited) ]OTU(Wrk_Alm);
   // This rung sets the Alarm (Alm) bit if the Input is true for the Minimum Duration time,
   // and sets (if Ack not required) or clears (if Ack required) the Acknowledge (Ack) bit
   // when the Alarm initially occurs, or when the Alarm is active and
   // becomes Enabled or Uninhibited.
   8: XIC(Inp)XIO(Disabled)XIO(Wrk_Inhibited)[TON(Wrk_MinDurationT,?,?) ,[XIC(Wrk_MinDurationT.DN) ,EQU(Wrk_MinDurationT.PRE,0) ] [XIO(Wrk_Alm) [XIC(Cfg_AckReqd) OTU(Ack) ,XIO(Cfg_AckReqd) OTL(Ack) ] ,OTL(Wrk_Alm) ] ];
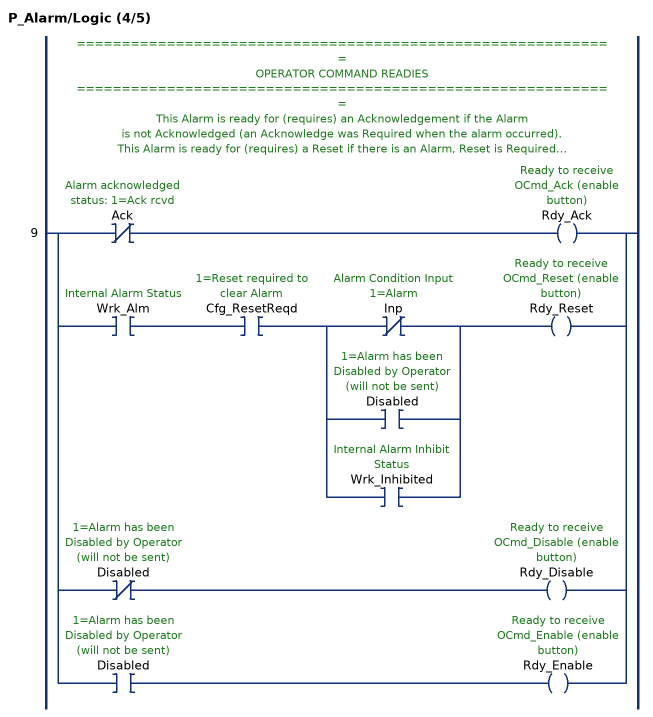
   // ============================================================
   // OPERATOR COMMAND READIES
   // ============================================================
   // This Alarm is ready for (requires) an Acknowledgement if the Alarm
   // is not Acknowledged (an Acknowledge was Required when the alarm occurred).
   // This Alarm is ready for (requires) a Reset if there is an Alarm, Reset is Required,
   // and the alarm condition has CLEARED.
   // If the Alarm is NOT Disabled, it is ready for Disable.
   // If the Alarm IS Disabled, it is ready for Enable.
   9: [XIO(Ack) OTE(Rdy_Ack) ,XIC(Wrk_Alm) XIC(Cfg_ResetReqd) [XIO(Inp) ,XIC(Disabled) ,XIC(Wrk_Inhibited) ] OTE(Rdy_Reset) ,XIO(Disabled) OTE(Rdy_Disable) ,XIC(Disabled) OTE(Rdy_Enable) ];
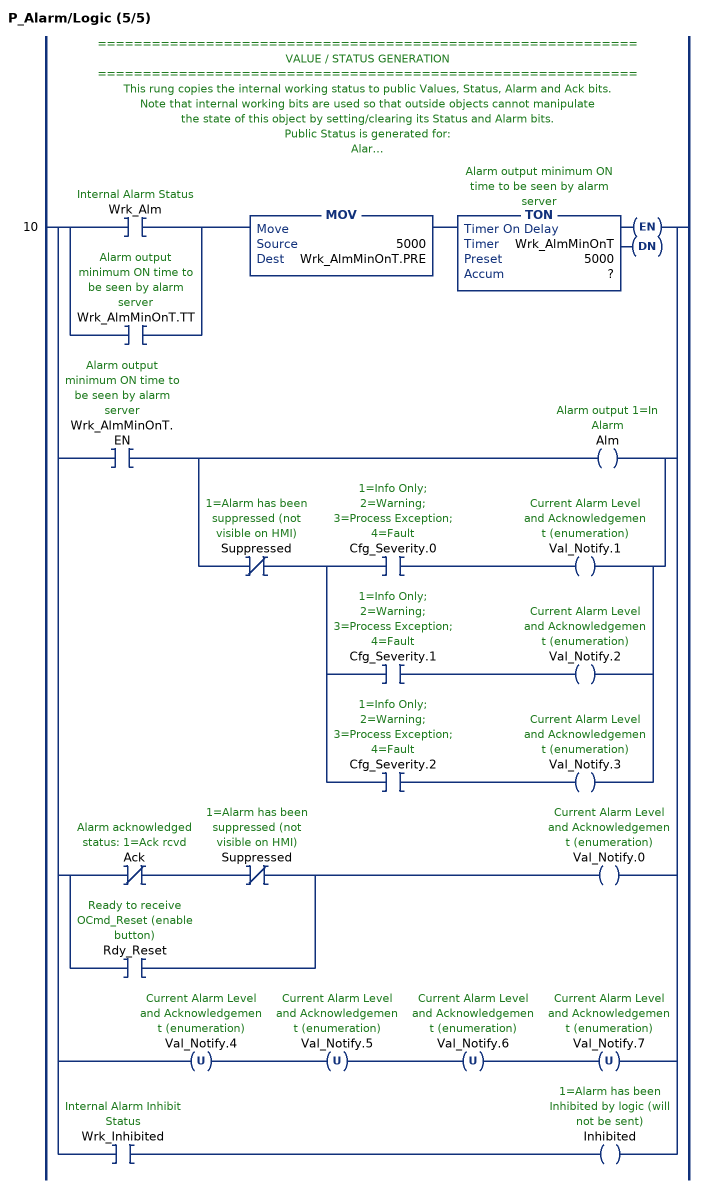
   // ============================================================
   // VALUE / STATUS GENERATION
   // ============================================================
   // This rung copies the internal working status to public Values, Status, Alarm and Ack bits.
   // Note that internal working bits are used so that outside objects cannot manipulate
   // the state of this object by setting/clearing its Status and Alarm bits.
   // Public Status is generated for:
   // Alarm
   // Notify Level (color, blink)
   // Alarm Inhibited
   // (Ack, Suppressed and Disabled can be set/cleared by the HMI directly.)
   10: [[XIC(Wrk_Alm) ,XIC(Wrk_AlmMinOnT.TT) ] MOV(5000,Wrk_AlmMinOnT.PRE) TON(Wrk_AlmMinOnT,?,?) ,XIC(Wrk_AlmMinOnT.EN) [OTE(Alm) ,XIO(Suppressed) [XIC(Cfg_Severity.0) OTE(Val_Notify.1) ,XIC(Cfg_Severity.1) OTE(Val_Notify.2) ,XIC(Cfg_Severity.2) OTE(Val_Notify.3) ] ] ,[XIO(Ack) XIO(Suppressed) ,XIC(Rdy_Reset) ] OTE(Val_Notify.0) ,OTU(Val_Notify.4) OTU(Val_Notify.5) OTU(Val_Notify.6) OTU(Val_Notify.7) ,XIC(Wrk_Inhibited) OTE(Inhibited) ];
END_ROUTINE
